% RSLogix 500 project DIGI PUMP CONTROL_BAK004.RSS, saved by version 8.30.00.16 %
PROJECT "AB"    % processor: Bul.1763 MicroLogix 1100 Series B %

PROGRAM FILES
  LAD 2 "MAIN"  3 rungs
  LAD 4 "DIGITAL_IO"  7 rungs
  LAD 5 "CONTROLS"  6 rungs

DATA FILES
  O0 OUTPUT  5 elements
  I1 INPUT  7 elements
  S2 STATUS  66 elements
  B3 BINARY  1 elements
  T4 TIMER  2 elements
  C5 COUNTER  1 elements
  R6 CONTROL  1 elements
  N7 INTEGER  1 elements
  F8 FLOAT  1 elements

LADDER 2 "MAIN"
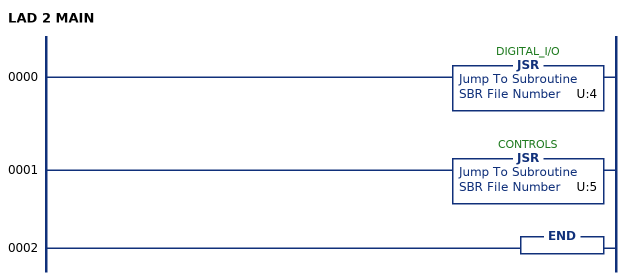
% Rung: 0 %
SOR JSR U:4 EOR
%   U:4  "DIGITAL_I/O" %
% Rung: 1 %
SOR JSR U:5 EOR
%   U:5  "CONTROLS" %
% Rung: 2 %
SOR END EOR

LADDER 4 "DIGITAL_IO"
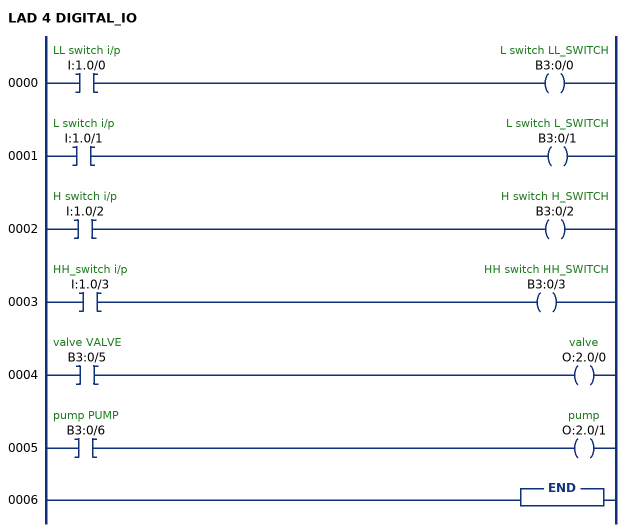
% Rung: 0 %
SOR XIC I:1.0/0 OTE B3:0/0 EOR
%   I:1.0/0  "LL switch i/p" %
%   B3:0/0  LL_SWITCH  "L switch" %
% Rung: 1 %
SOR XIC I:1.0/1 OTE B3:0/1 EOR
%   I:1.0/1  "L switch i/p" %
%   B3:0/1  L_SWITCH  "L switch" %
% Rung: 2 %
SOR XIC I:1.0/2 OTE B3:0/2 EOR
%   I:1.0/2  "H switch i/p" %
%   B3:0/2  H_SWITCH  "H switch" %
% Rung: 3 %
SOR XIC I:1.0/3 OTE B3:0/3 EOR
%   I:1.0/3  "HH_switch i/p" %
%   B3:0/3  HH_SWITCH  "HH switch" %
% Rung: 4 %
SOR XIC B3:0/5 OTE O:2.0/0 EOR
%   B3:0/5  VALVE  "valve" %
%   O:2.0/0  "valve" %
% Rung: 5 %
SOR XIC B3:0/6 OTE O:2.0/1 EOR
%   B3:0/6  PUMP  "pump" %
%   O:2.0/1  "pump" %
% Rung: 6 %
SOR END EOR

LADDER 5 "CONTROLS"
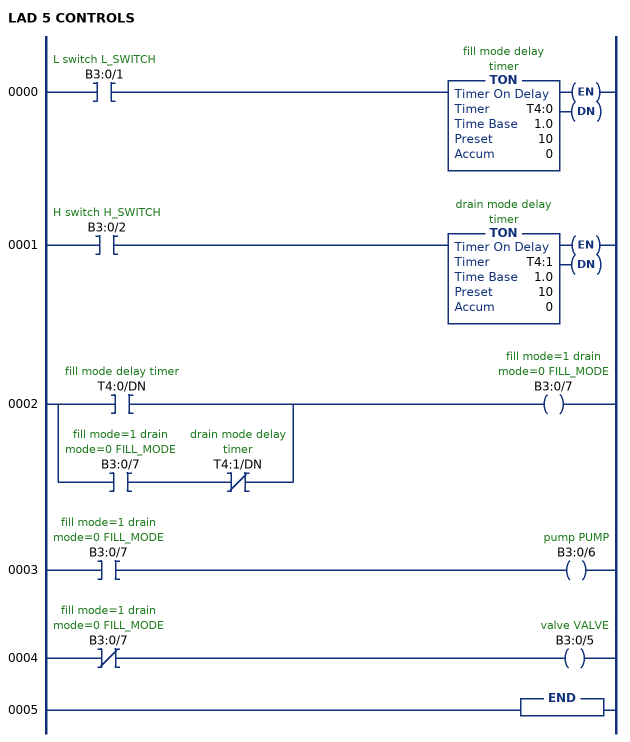
% Rung: 0 %
SOR XIC B3:0/1 TON T4:0 1.0 10 0 EOR
%   B3:0/1  L_SWITCH  "L switch" %
%   T4:0  "fill mode delay timer" %
% Rung: 1 %
SOR XIC B3:0/2 TON T4:1 1.0 10 0 EOR
%   B3:0/2  H_SWITCH  "H switch" %
%   T4:1  "drain mode delay timer" %
% Rung: 2 %
SOR BST XIC T4:0/DN NXB XIC B3:0/7 XIO T4:1/DN BND OTE B3:0/7 EOR
%   T4:0/DN  "fill mode delay timer" %
%   B3:0/7  FILL_MODE  "fill mode=1 drain mode=0" %
%   T4:1/DN  "drain mode delay timer" %
% Rung: 3 %
SOR XIC B3:0/7 OTE B3:0/6 EOR
%   B3:0/7  FILL_MODE  "fill mode=1 drain mode=0" %
%   B3:0/6  PUMP  "pump" %
% Rung: 4 %
SOR XIO B3:0/7 OTE B3:0/5 EOR
%   B3:0/7  FILL_MODE  "fill mode=1 drain mode=0" %
%   B3:0/5  VALVE  "valve" %
% Rung: 5 %
SOR END EOR

DATA TABLE (non-zero values as saved)
DATA T4
% .PRE .ACC %
% T4:0 % 10 0
% T4:1 % 10 0
